FUNCTION_BLOCK FB_NE_COLOR (* Test for COLOR Inequality *)
  (* Standard: 61499-1 *)
  (* Version 0.1, 2004096-21, JHC, Rockwell Automation, Moved from hmi to math. *)
  (* Version 0.0, 2001-04-05, JHC, Rockwell Automation, First XML version. *)
  (* Compiler header: package fb.rt.math; *)
  (* Compiler Java Sun JDK 1.4.2 *)
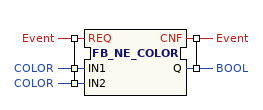
  EVENT_INPUT
    REQ WITH IN1, IN2;
  END_EVENT
  EVENT_OUTPUT
    CNF WITH Q;
  END_EVENT
  VAR_INPUT
    IN1 : COLOR;
    IN2 : COLOR;
  END_VAR
  VAR_OUTPUT
    Q : BOOL; (* IN1<>IN2 *)
  END_VAR
END_FUNCTION_BLOCK
